% RSLogix 500 project I2P Job 12B - Myah.RSS, saved by version 10.00.00.00 %
PROJECT "ML05B"    % processor: Bul.1763 MicroLogix 1100 Series B %

PROGRAM FILES
  LAD 2   11 rungs

DATA FILES
  O0 OUTPUT  4 elements
  I1 INPUT  6 elements
  S2 STATUS  66 elements
  B3 BINARY  1 elements
  T4 TIMER  1 elements
  C5 COUNTER  1 elements
  R6 CONTROL  1 elements
  N7 INTEGER  1 elements
  F8 FLOAT  1 elements

LADDER 2
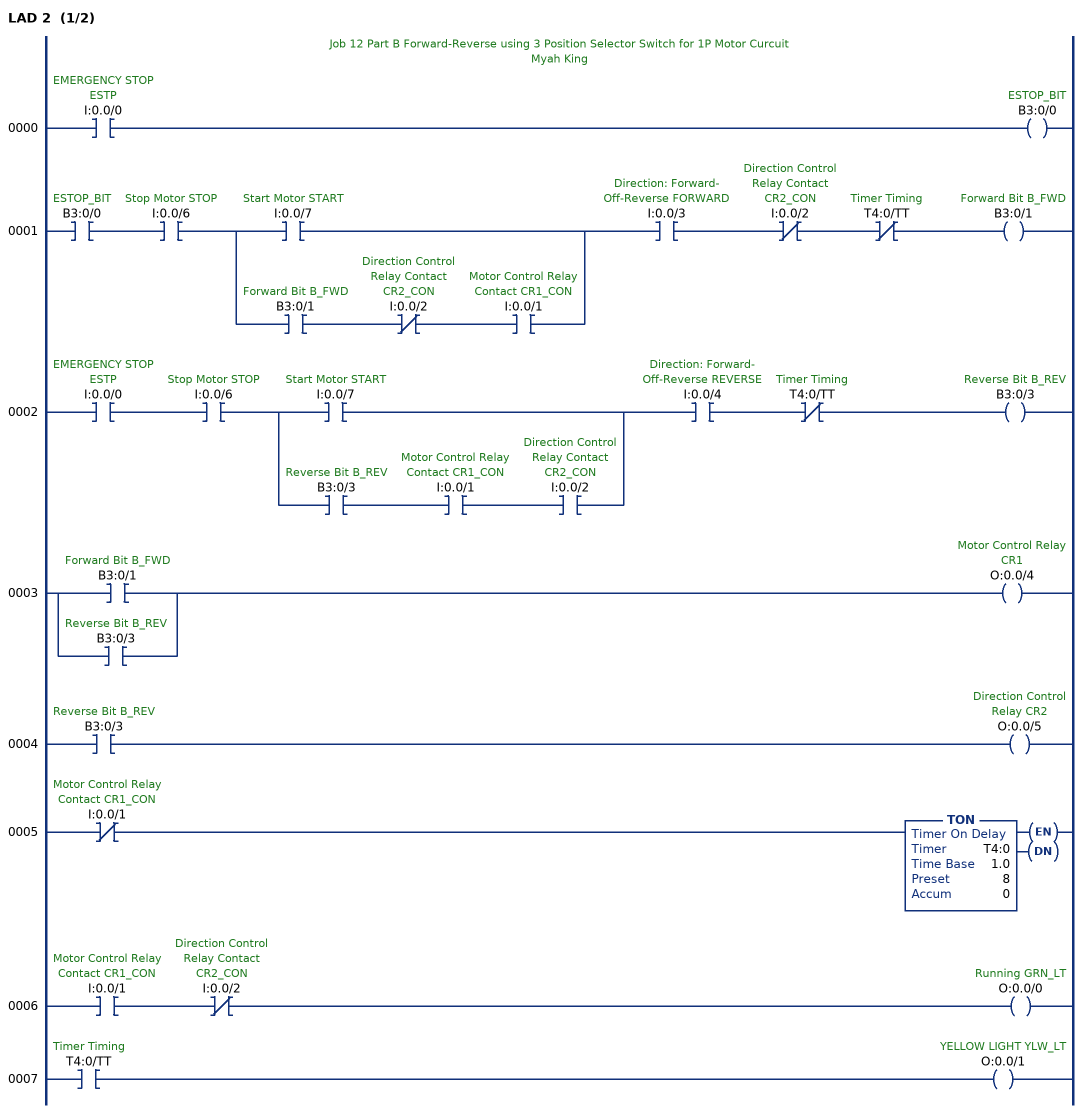
% Rung: 0 %
% Job 12 Part B Forward-Reverse using 3 Position Selector Switch for 1P Motor Curcuit
% Myah King %
SOR XIC I:0.0/0 OTE B3:0/0 EOR
%   I:0.0/0  ESTP  "EMERGENCY STOP" %
%   B3:0/0  ESTOP_BIT %
% Rung: 1 %
SOR XIC B3:0/0 XIC I:0.0/6 BST XIC I:0.0/7 NXB XIC B3:0/1 XIO I:0.0/2 XIC I:0.0/1 BND XIC I:0.0/3 XIO I:0.0/2 XIO T4:0/TT OTE B3:0/1 EOR
%   B3:0/0  ESTOP_BIT %
%   I:0.0/6  STOP  "Stop Motor" %
%   I:0.0/7  START  "Start Motor" %
%   B3:0/1  B_FWD  "Forward Bit" %
%   I:0.0/2  CR2_CON  "Direction Control Relay Contact" %
%   I:0.0/1  CR1_CON  "Motor Control Relay Contact" %
%   I:0.0/3  FORWARD  "Direction: Forward- Off-Reverse" %
%   T4:0/TT  "Timer Timing" %
% Rung: 2 %
SOR XIC I:0.0/0 XIC I:0.0/6 BST XIC I:0.0/7 NXB XIC B3:0/3 XIC I:0.0/1 XIC I:0.0/2 BND XIC I:0.0/4 XIO T4:0/TT OTE B3:0/3 EOR
%   I:0.0/0  ESTP  "EMERGENCY STOP" %
%   I:0.0/6  STOP  "Stop Motor" %
%   I:0.0/7  START  "Start Motor" %
%   B3:0/3  B_REV  "Reverse Bit" %
%   I:0.0/1  CR1_CON  "Motor Control Relay Contact" %
%   I:0.0/2  CR2_CON  "Direction Control Relay Contact" %
%   I:0.0/4  REVERSE  "Direction: Forward- Off-Reverse" %
%   T4:0/TT  "Timer Timing" %
% Rung: 3 %
SOR BST XIC B3:0/1 NXB XIC B3:0/3 BND OTE O:0.0/4 EOR
%   B3:0/1  B_FWD  "Forward Bit" %
%   B3:0/3  B_REV  "Reverse Bit" %
%   O:0.0/4  CR1  "Motor Control Relay" %
% Rung: 4 %
SOR XIC B3:0/3 OTE O:0.0/5 EOR
%   B3:0/3  B_REV  "Reverse Bit" %
%   O:0.0/5  CR2  "Direction Control Relay" %
% Rung: 5 %
SOR XIO I:0.0/1 TON T4:0 1.0 8 0 EOR
%   I:0.0/1  CR1_CON  "Motor Control Relay Contact" %
% Rung: 6 %
SOR XIC I:0.0/1 XIO I:0.0/2 OTE O:0.0/0 EOR
%   I:0.0/1  CR1_CON  "Motor Control Relay Contact" %
%   I:0.0/2  CR2_CON  "Direction Control Relay Contact" %
%   O:0.0/0  GRN_LT  "Running" %
% Rung: 7 %
SOR XIC T4:0/TT OTE O:0.0/1 EOR
%   T4:0/TT  "Timer Timing" %
%   O:0.0/1  YLW_LT  "YELLOW LIGHT" %

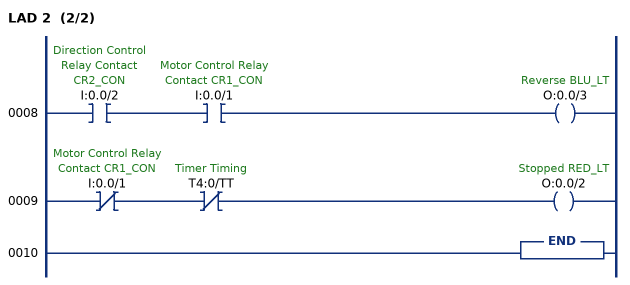
% Rung: 8 %
SOR XIC I:0.0/2 XIC I:0.0/1 OTE O:0.0/3 EOR
%   I:0.0/2  CR2_CON  "Direction Control Relay Contact" %
%   I:0.0/1  CR1_CON  "Motor Control Relay Contact" %
%   O:0.0/3  BLU_LT  "Reverse" %
% Rung: 9 %
SOR XIO I:0.0/1 XIO T4:0/TT OTE O:0.0/2 EOR
%   I:0.0/1  CR1_CON  "Motor Control Relay Contact" %
%   T4:0/TT  "Timer Timing" %
%   O:0.0/2  RED_LT  "Stopped" %
% Rung: 10 %
SOR END EOR

OTHER DOCUMENTED ADDRESSES
  I:0.0/5  2PSS  "2 POSITION SELECTOR SWITCH"
  I:0.0/8  JOG  "NORMALLY OPEN PUSH BUTTON 2"

DATA TABLE (non-zero values as saved)
DATA B3
% B3:0 % 0X0001
DATA T4
% .PRE .ACC %
% T4:0 % 8 0
